DATA_BLOCK "InstGetIdentMv"   // DB220
// stored: InstanceOfName GetIdentMv, InstanceOfType FB
"GetIdentMv"
BEGIN
   identMvAllUnits[0].identMvEM[0..7].selectedUnit := 0;
   identMvAllUnits[0].identMvEM[0..7].selectedEM := 0;
   identMvAllUnits[0].identMvEM[0..7].mvReaderId := 0;
   identMvAllUnits[0].identMvEM[0..7].numberOfMv := 0;
   identMvAllUnits[0].identMvEM[0].mvReader[0..1].deviceName := WSTRING#'';
   identMvAllUnits[0].identMvEM[1].mvReader[0..1].deviceName := WSTRING#'';
   identMvAllUnits[0].identMvEM[2].mvReader[0..1].deviceName := WSTRING#'';
   identMvAllUnits[0].identMvEM[3].mvReader[0..1].deviceName := WSTRING#'';
   identMvAllUnits[0].identMvEM[4].mvReader[0..1].deviceName := WSTRING#'';
   identMvAllUnits[0].identMvEM[5].mvReader[0..1].deviceName := WSTRING#'';
   identMvAllUnits[0].identMvEM[6].mvReader[0..1].deviceName := WSTRING#'';
   identMvAllUnits[0].identMvEM[7].mvReader[0..1].deviceName := WSTRING#'';
   identMvAllUnits[0].identMvEM[0].mvReader[0..1].deviceType := WSTRING#'';
   identMvAllUnits[0].identMvEM[1].mvReader[0..1].deviceType := WSTRING#'';
   identMvAllUnits[0].identMvEM[2].mvReader[0..1].deviceType := WSTRING#'';
   identMvAllUnits[0].identMvEM[3].mvReader[0..1].deviceType := WSTRING#'';
   identMvAllUnits[0].identMvEM[4].mvReader[0..1].deviceType := WSTRING#'';
   identMvAllUnits[0].identMvEM[5].mvReader[0..1].deviceType := WSTRING#'';
   identMvAllUnits[0].identMvEM[6].mvReader[0..1].deviceType := WSTRING#'';
   identMvAllUnits[0].identMvEM[7].mvReader[0..1].deviceType := WSTRING#'';
   identMvAllUnits[0].identMvEM[0].mvReader[0..1].deviceId := 0;
   identMvAllUnits[0].identMvEM[1].mvReader[0..1].deviceId := 0;
   identMvAllUnits[0].identMvEM[2].mvReader[0..1].deviceId := 0;
   identMvAllUnits[0].identMvEM[3].mvReader[0..1].deviceId := 0;
   identMvAllUnits[0].identMvEM[4].mvReader[0..1].deviceId := 0;
   identMvAllUnits[0].identMvEM[5].mvReader[0..1].deviceId := 0;
   identMvAllUnits[0].identMvEM[6].mvReader[0..1].deviceId := 0;
   identMvAllUnits[0].identMvEM[7].mvReader[0..1].deviceId := 0;
   identMvAllUnits[0].identMvEM[0].mvReader[0..1].tagType := WSTRING#'';
   identMvAllUnits[0].identMvEM[1].mvReader[0..1].tagType := WSTRING#'';
   identMvAllUnits[0].identMvEM[2].mvReader[0..1].tagType := WSTRING#'';
   identMvAllUnits[0].identMvEM[3].mvReader[0..1].tagType := WSTRING#'';
   identMvAllUnits[0].identMvEM[4].mvReader[0..1].tagType := WSTRING#'';
   identMvAllUnits[0].identMvEM[5].mvReader[0..1].tagType := WSTRING#'';
   identMvAllUnits[0].identMvEM[6].mvReader[0..1].tagType := WSTRING#'';
   identMvAllUnits[0].identMvEM[7].mvReader[0..1].tagType := WSTRING#'';
   identMvAllUnits[0].identMvEM[0].mvReader[0..1].cameraMode := WSTRING#'';
   identMvAllUnits[0].identMvEM[1].mvReader[0..1].cameraMode := WSTRING#'';
   identMvAllUnits[0].identMvEM[2].mvReader[0..1].cameraMode := WSTRING#'';
   identMvAllUnits[0].identMvEM[3].mvReader[0..1].cameraMode := WSTRING#'';
   identMvAllUnits[0].identMvEM[4].mvReader[0..1].cameraMode := WSTRING#'';
   identMvAllUnits[0].identMvEM[5].mvReader[0..1].cameraMode := WSTRING#'';
   identMvAllUnits[0].identMvEM[6].mvReader[0..1].cameraMode := WSTRING#'';
   identMvAllUnits[0].identMvEM[7].mvReader[0..1].cameraMode := WSTRING#'';
   identMvAllUnits[0].identMvEM[0].mvReader[0..1].resultState := WSTRING#'';
   identMvAllUnits[0].identMvEM[1].mvReader[0..1].resultState := WSTRING#'';
   identMvAllUnits[0].identMvEM[2].mvReader[0..1].resultState := WSTRING#'';
   identMvAllUnits[0].identMvEM[3].mvReader[0..1].resultState := WSTRING#'';
   identMvAllUnits[0].identMvEM[4].mvReader[0..1].resultState := WSTRING#'';
   identMvAllUnits[0].identMvEM[5].mvReader[0..1].resultState := WSTRING#'';
   identMvAllUnits[0].identMvEM[6].mvReader[0..1].resultState := WSTRING#'';
   identMvAllUnits[0].identMvEM[7].mvReader[0..1].resultState := WSTRING#'';
   identMvAllUnits[0].identMvEM[0].mvReader[0..1].progNo := 0;
   identMvAllUnits[0].identMvEM[1].mvReader[0..1].progNo := 0;
   identMvAllUnits[0].identMvEM[2].mvReader[0..1].progNo := 0;
   identMvAllUnits[0].identMvEM[3].mvReader[0..1].progNo := 0;
   identMvAllUnits[0].identMvEM[4].mvReader[0..1].progNo := 0;
   identMvAllUnits[0].identMvEM[5].mvReader[0..1].progNo := 0;
   identMvAllUnits[0].identMvEM[6].mvReader[0..1].progNo := 0;
   identMvAllUnits[0].identMvEM[7].mvReader[0..1].progNo := 0;
   identMvAllUnits[0].identMvEM[0].mvReader[0..1].progNumberWrite := 0;
   identMvAllUnits[0].identMvEM[1].mvReader[0..1].progNumberWrite := 0;
   identMvAllUnits[0].identMvEM[2].mvReader[0..1].progNumberWrite := 0;
   identMvAllUnits[0].identMvEM[3].mvReader[0..1].progNumberWrite := 0;
   identMvAllUnits[0].identMvEM[4].mvReader[0..1].progNumberWrite := 0;
   identMvAllUnits[0].identMvEM[5].mvReader[0..1].progNumberWrite := 0;
   identMvAllUnits[0].identMvEM[6].mvReader[0..1].progNumberWrite := 0;
   identMvAllUnits[0].identMvEM[7].mvReader[0..1].progNumberWrite := 0;
   identMvAllUnits[0].identMvEM[0].mvReader[0..1].pushbutton := 16#0000;
   identMvAllUnits[0].identMvEM[1].mvReader[0..1].pushbutton := 16#0000;
   identMvAllUnits[0].identMvEM[2].mvReader[0..1].pushbutton := 16#0000;
   identMvAllUnits[0].identMvEM[3].mvReader[0..1].pushbutton := 16#0000;
   identMvAllUnits[0].identMvEM[4].mvReader[0..1].pushbutton := 16#0000;
   identMvAllUnits[0].identMvEM[5].mvReader[0..1].pushbutton := 16#0000;
   identMvAllUnits[0].identMvEM[6].mvReader[0..1].pushbutton := 16#0000;
   identMvAllUnits[0].identMvEM[7].mvReader[0..1].pushbutton := 16#0000;
   identMvAllUnits[0].identMvEM[0].mvReader[0..1].enablePushbutton := 16#0000;
   identMvAllUnits[0].identMvEM[1].mvReader[0..1].enablePushbutton := 16#0000;
   identMvAllUnits[0].identMvEM[2].mvReader[0..1].enablePushbutton := 16#0000;
   identMvAllUnits[0].identMvEM[3].mvReader[0..1].enablePushbutton := 16#0000;
   identMvAllUnits[0].identMvEM[4].mvReader[0..1].enablePushbutton := 16#0000;
   identMvAllUnits[0].identMvEM[5].mvReader[0..1].enablePushbutton := 16#0000;
   identMvAllUnits[0].identMvEM[6].mvReader[0..1].enablePushbutton := 16#0000;
   identMvAllUnits[0].identMvEM[7].mvReader[0..1].enablePushbutton := 16#0000;
   identMvAllUnits[0].identMvEM[0].mvReader[0..1].status := 16#0000;
   identMvAllUnits[0].identMvEM[1].mvReader[0..1].status := 16#0000;
   identMvAllUnits[0].identMvEM[2].mvReader[0..1].status := 16#0000;
   identMvAllUnits[0].identMvEM[3].mvReader[0..1].status := 16#0000;
   identMvAllUnits[0].identMvEM[4].mvReader[0..1].status := 16#0000;
   identMvAllUnits[0].identMvEM[5].mvReader[0..1].status := 16#0000;
   identMvAllUnits[0].identMvEM[6].mvReader[0..1].status := 16#0000;
   identMvAllUnits[0].identMvEM[7].mvReader[0..1].status := 16#0000;
   identMvAllUnits[0].identMvEM[0].mvReader[0..1].alarmCategorie := 0;
   identMvAllUnits[0].identMvEM[1].mvReader[0..1].alarmCategorie := 0;
   identMvAllUnits[0].identMvEM[2].mvReader[0..1].alarmCategorie := 0;
   identMvAllUnits[0].identMvEM[3].mvReader[0..1].alarmCategorie := 0;
   identMvAllUnits[0].identMvEM[4].mvReader[0..1].alarmCategorie := 0;
   identMvAllUnits[0].identMvEM[5].mvReader[0..1].alarmCategorie := 0;
   identMvAllUnits[0].identMvEM[6].mvReader[0..1].alarmCategorie := 0;
   identMvAllUnits[0].identMvEM[7].mvReader[0..1].alarmCategorie := 0;
   identMvAllUnits[0].identMvEM[0].mvReader[0..1].alarmNo := 0;
   identMvAllUnits[0].identMvEM[1].mvReader[0..1].alarmNo := 0;
   identMvAllUnits[0].identMvEM[2].mvReader[0..1].alarmNo := 0;
   identMvAllUnits[0].identMvEM[3].mvReader[0..1].alarmNo := 0;
   identMvAllUnits[0].identMvEM[4].mvReader[0..1].alarmNo := 0;
   identMvAllUnits[0].identMvEM[5].mvReader[0..1].alarmNo := 0;
   identMvAllUnits[0].identMvEM[6].mvReader[0..1].alarmNo := 0;
   identMvAllUnits[0].identMvEM[7].mvReader[0..1].alarmNo := 0;
   identMvAllUnits[0].identMvEM[0].mvReader[0..1].alarmCode := 16#0000_0000;
   identMvAllUnits[0].identMvEM[1].mvReader[0..1].alarmCode := 16#0000_0000;
   identMvAllUnits[0].identMvEM[2].mvReader[0..1].alarmCode := 16#0000_0000;
   identMvAllUnits[0].identMvEM[3].mvReader[0..1].alarmCode := 16#0000_0000;
   identMvAllUnits[0].identMvEM[4].mvReader[0..1].alarmCode := 16#0000_0000;
   identMvAllUnits[0].identMvEM[5].mvReader[0..1].alarmCode := 16#0000_0000;
   identMvAllUnits[0].identMvEM[6].mvReader[0..1].alarmCode := 16#0000_0000;
   identMvAllUnits[0].identMvEM[7].mvReader[0..1].alarmCode := 16#0000_0000;
   identMvAllUnits[0].identMvEM[0].mvReader[0..1].resultColor := 0;
   identMvAllUnits[0].identMvEM[1].mvReader[0..1].resultColor := 0;
   identMvAllUnits[0].identMvEM[2].mvReader[0..1].resultColor := 0;
   identMvAllUnits[0].identMvEM[3].mvReader[0..1].resultColor := 0;
   identMvAllUnits[0].identMvEM[4].mvReader[0..1].resultColor := 0;
   identMvAllUnits[0].identMvEM[5].mvReader[0..1].resultColor := 0;
   identMvAllUnits[0].identMvEM[6].mvReader[0..1].resultColor := 0;
   identMvAllUnits[0].identMvEM[7].mvReader[0..1].resultColor := 0;
   identMvAllUnits[0].identMvEM[0].mvReader[0..1].statusColorCode := 0;
   identMvAllUnits[0].identMvEM[1].mvReader[0..1].statusColorCode := 0;
   identMvAllUnits[0].identMvEM[2].mvReader[0..1].statusColorCode := 0;
   identMvAllUnits[0].identMvEM[3].mvReader[0..1].statusColorCode := 0;
   identMvAllUnits[0].identMvEM[4].mvReader[0..1].statusColorCode := 0;
   identMvAllUnits[0].identMvEM[5].mvReader[0..1].statusColorCode := 0;
   identMvAllUnits[0].identMvEM[6].mvReader[0..1].statusColorCode := 0;
   identMvAllUnits[0].identMvEM[7].mvReader[0..1].statusColorCode := 0;
   identMvAllUnits[0].identMvEM[0].mvReader[0..1].datRead1 := '';
   identMvAllUnits[0].identMvEM[1].mvReader[0..1].datRead1 := '';
   identMvAllUnits[0].identMvEM[2].mvReader[0..1].datRead1 := '';
   identMvAllUnits[0].identMvEM[3].mvReader[0..1].datRead1 := '';
   identMvAllUnits[0].identMvEM[4].mvReader[0..1].datRead1 := '';
   identMvAllUnits[0].identMvEM[5].mvReader[0..1].datRead1 := '';
   identMvAllUnits[0].identMvEM[6].mvReader[0..1].datRead1 := '';
   identMvAllUnits[0].identMvEM[7].mvReader[0..1].datRead1 := '';
   identMvAllUnits[0].identMvEM[0].mvReader[0..1].datRead2 := '';
   identMvAllUnits[0].identMvEM[1].mvReader[0..1].datRead2 := '';
   identMvAllUnits[0].identMvEM[2].mvReader[0..1].datRead2 := '';
   identMvAllUnits[0].identMvEM[3].mvReader[0..1].datRead2 := '';
   identMvAllUnits[0].identMvEM[4].mvReader[0..1].datRead2 := '';
   identMvAllUnits[0].identMvEM[5].mvReader[0..1].datRead2 := '';
   identMvAllUnits[0].identMvEM[6].mvReader[0..1].datRead2 := '';
   identMvAllUnits[0].identMvEM[7].mvReader[0..1].datRead2 := '';
   identMvAllUnits[0].identMvEM[0].mvReader[0..1].datRead3 := '';
   identMvAllUnits[0].identMvEM[1].mvReader[0..1].datRead3 := '';
   identMvAllUnits[0].identMvEM[2].mvReader[0..1].datRead3 := '';
   identMvAllUnits[0].identMvEM[3].mvReader[0..1].datRead3 := '';
   identMvAllUnits[0].identMvEM[4].mvReader[0..1].datRead3 := '';
   identMvAllUnits[0].identMvEM[5].mvReader[0..1].datRead3 := '';
   identMvAllUnits[0].identMvEM[6].mvReader[0..1].datRead3 := '';
   identMvAllUnits[0].identMvEM[7].mvReader[0..1].datRead3 := '';
   identMvAllUnits[0].identMvEM[0].mvReader[0..1].datRead4 := '';
   identMvAllUnits[0].identMvEM[1].mvReader[0..1].datRead4 := '';
   identMvAllUnits[0].identMvEM[2].mvReader[0..1].datRead4 := '';
   identMvAllUnits[0].identMvEM[3].mvReader[0..1].datRead4 := '';
   identMvAllUnits[0].identMvEM[4].mvReader[0..1].datRead4 := '';
   identMvAllUnits[0].identMvEM[5].mvReader[0..1].datRead4 := '';
   identMvAllUnits[0].identMvEM[6].mvReader[0..1].datRead4 := '';
   identMvAllUnits[0].identMvEM[7].mvReader[0..1].datRead4 := '';
   identMvAllUnits[0].identMvEM[0].mvReader[0].datWrite1 := '';
   identMvAllUnits[0].identMvEM[0].mvReader[1].datWrite1 := 'Siemens';
   identMvAllUnits[0].identMvEM[1].mvReader[0..1].datWrite1 := '';
   identMvAllUnits[0].identMvEM[2].mvReader[0..1].datWrite1 := '';
   identMvAllUnits[0].identMvEM[3].mvReader[0..1].datWrite1 := '';
   identMvAllUnits[0].identMvEM[4].mvReader[0..1].datWrite1 := '';
   identMvAllUnits[0].identMvEM[5].mvReader[0..1].datWrite1 := '';
   identMvAllUnits[0].identMvEM[6].mvReader[0..1].datWrite1 := '';
   identMvAllUnits[0].identMvEM[7].mvReader[0..1].datWrite1 := '';
   identMvAllUnits[0].identMvEM[0].mvReader[0..1].datWrite2 := '';
   identMvAllUnits[0].identMvEM[1].mvReader[0..1].datWrite2 := '';
   identMvAllUnits[0].identMvEM[2].mvReader[0..1].datWrite2 := '';
   identMvAllUnits[0].identMvEM[3].mvReader[0..1].datWrite2 := '';
   identMvAllUnits[0].identMvEM[4].mvReader[0..1].datWrite2 := '';
   identMvAllUnits[0].identMvEM[5].mvReader[0..1].datWrite2 := '';
   identMvAllUnits[0].identMvEM[6].mvReader[0..1].datWrite2 := '';
   identMvAllUnits[0].identMvEM[7].mvReader[0..1].datWrite2 := '';
   identMvAllUnits[0].identMvEM[0].mvReader[0..1].datWrite3 := '';
   identMvAllUnits[0].identMvEM[1].mvReader[0..1].datWrite3 := '';
   identMvAllUnits[0].identMvEM[2].mvReader[0..1].datWrite3 := '';
   identMvAllUnits[0].identMvEM[3].mvReader[0..1].datWrite3 := '';
   identMvAllUnits[0].identMvEM[4].mvReader[0..1].datWrite3 := '';
   identMvAllUnits[0].identMvEM[5].mvReader[0..1].datWrite3 := '';
   identMvAllUnits[0].identMvEM[6].mvReader[0..1].datWrite3 := '';
   identMvAllUnits[0].identMvEM[7].mvReader[0..1].datWrite3 := '';
   identMvAllUnits[0].identMvEM[0].mvReader[0..1].datWrite4 := '';
   identMvAllUnits[0].identMvEM[1].mvReader[0..1].datWrite4 := '';
   identMvAllUnits[0].identMvEM[2].mvReader[0..1].datWrite4 := '';
   identMvAllUnits[0].identMvEM[3].mvReader[0..1].datWrite4 := '';
   identMvAllUnits[0].identMvEM[4].mvReader[0..1].datWrite4 := '';
   identMvAllUnits[0].identMvEM[5].mvReader[0..1].datWrite4 := '';
   identMvAllUnits[0].identMvEM[6].mvReader[0..1].datWrite4 := '';
   identMvAllUnits[0].identMvEM[7].mvReader[0..1].datWrite4 := '';
END_DATA_BLOCK

DATA_BLOCK "Et200SpMotorstarterInterfaceHmi"   // DB208
// stored: InstanceOfName typeEt200SpMotorstarterInterfaceHmi, InstanceOfType UDT
"typeEt200SpMotorstarterInterfaceHmi"
BEGIN
   et200SpMotorstarterCurrent[0..1] := 0.0;
   et200SpMotorstarterInputs[0..1].readyAutomatic := FALSE;
   et200SpMotorstarterInputs[0..1].motorOn := FALSE;
   et200SpMotorstarterInputs[0..1].groupFault := FALSE;
   et200SpMotorstarterInputs[0..1].groupWarning := FALSE;
   et200SpMotorstarterInputs[0..1].input1 := FALSE;
   et200SpMotorstarterInputs[0..1].input2 := FALSE;
   et200SpMotorstarterInputs[0..1].input3 := FALSE;
   et200SpMotorstarterInputs[0..1].inputLocalCtrl := FALSE;
   et200SpMotorstarterInputs[0..1].iActBit0 := FALSE;
   et200SpMotorstarterInputs[0..1].iActBit1 := FALSE;
   et200SpMotorstarterInputs[0..1].iActBit2 := FALSE;
   et200SpMotorstarterInputs[0..1].iActBit3 := FALSE;
   et200SpMotorstarterInputs[0..1].iActBit4 := FALSE;
   et200SpMotorstarterInputs[0..1].iActBit5 := FALSE;
   et200SpMotorstarterInputs[0..1].manualOperating := FALSE;
   et200SpMotorstarterInputs[0..1].spare1 := FALSE;
   et200SpMotorstarterInputs[0..1].readyStartOn := FALSE;
   et200SpMotorstarterInputs[0..1].motorOnRight := FALSE;
   et200SpMotorstarterInputs[0..1].motorOnLeft := FALSE;
   et200SpMotorstarterInputs[0..1].quickstopActive := FALSE;
   et200SpMotorstarterInputs[0..1].energySaving := FALSE;
   et200SpMotorstarterInputs[0..1].moduleInserted := FALSE;
   et200SpMotorstarterInputs[0..1].exProtectionMotorActive := FALSE;
   et200SpMotorstarterInputs[0..1].blockActive := FALSE;
   et200SpMotorstarterInputs[0..1].thermalMotorOverload := FALSE;
   et200SpMotorstarterInputs[0..1].spare5 := FALSE;
   et200SpMotorstarterInputs[0..1].currentLimitTripping := FALSE;
   et200SpMotorstarterInputs[0..1].statusFailDi := FALSE;
   et200SpMotorstarterInputs[0..1].residualCurrent := FALSE;
   et200SpMotorstarterInputs[0..1].asymmetryDetected := FALSE;
   et200SpMotorstarterInputs[0..1].overtemperature := FALSE;
   et200SpMotorstarterInputs[0..1].spare7 := FALSE;
   et200SpMotorstarterOutputs[0..1].motorCw := FALSE;
   et200SpMotorstarterOutputs[0..1].motorCww := FALSE;
   et200SpMotorstarterOutputs[0..1].reserve1 := FALSE;
   et200SpMotorstarterOutputs[0..1].tripReset := FALSE;
   et200SpMotorstarterOutputs[0..1].emergencyStart := FALSE;
   et200SpMotorstarterOutputs[0..1].reserve2 := FALSE;
   et200SpMotorstarterOutputs[0..1].reserve3 := FALSE;
   et200SpMotorstarterOutputs[0..1].coldStart := FALSE;
   et200SpMotorstarterOutputs[0..1].reserve4 := FALSE;
   et200SpMotorstarterOutputs[0..1].reserve5 := FALSE;
   et200SpMotorstarterOutputs[0..1].reserve6 := FALSE;
   et200SpMotorstarterOutputs[0..1].reserve7 := FALSE;
   et200SpMotorstarterOutputs[0..1].reserve8 := FALSE;
   et200SpMotorstarterOutputs[0..1].reserve9 := FALSE;
   et200SpMotorstarterOutputs[0..1].reserve10 := FALSE;
   et200SpMotorstarterOutputs[0..1].disableQuickStop := FALSE;
END_DATA_BLOCK
